afAl[0  , 0] := 1.00000E+01; afAl[0  , 1] := 2.70842E-02;
afAl[1  , 0] := 1.99800E+01; afAl[1  , 1] := 3.60106E-02;
afAl[2  , 0] := 2.99600E+01; afAl[2  , 1] := 1.04693E-01;
afAl[3  , 0] := 3.99400E+01; afAl[3  , 1] := 1.64797E-01;
afAl[4  , 0] := 4.99200E+01; afAl[4  , 1] := 1.89347E-01;
afAl[5  , 0] := 5.99000E+01; afAl[5  , 1] := 1.90141E-01;
afAl[6  , 0] := 6.98800E+01; afAl[6  , 1] := 1.82197E-01;
afAl[7  , 0] := 7.98600E+01; afAl[7  , 1] := 5.02769E+00;
afAl[8  , 0] := 8.98400E+01; afAl[8  , 1] := 6.70542E+00;
afAl[9  , 0] := 9.98200E+01; afAl[9  , 1] := 7.82345E+00;
afAl[10 , 0] := 1.09800E+02; afAl[10 , 1] := 8.42194E+00;
afAl[11 , 0] := 1.19780E+02; afAl[11 , 1] := 9.34640E+00;
afAl[12 , 0] := 1.29760E+02; afAl[12 , 1] := 9.38873E+00;
afAl[13 , 0] := 1.39740E+02; afAl[13 , 1] := 9.18537E+00;
afAl[14 , 0] := 1.49720E+02; afAl[14 , 1] := 8.86987E+00;
afAl[15 , 0] := 1.59700E+02; afAl[15 , 1] := 8.49608E+00;
afAl[16 , 0] := 1.69680E+02; afAl[16 , 1] := 8.09707E+00;
afAl[17 , 0] := 1.79660E+02; afAl[17 , 1] := 7.69477E+00;
afAl[18 , 0] := 1.89640E+02; afAl[18 , 1] := 7.30166E+00;
afAl[19 , 0] := 1.99620E+02; afAl[19 , 1] := 6.92482E+00;
afAl[20 , 0] := 2.09600E+02; afAl[20 , 1] := 6.56777E+00;
afAl[21 , 0] := 2.19580E+02; afAl[21 , 1] := 6.23207E+00;
afAl[22 , 0] := 2.29560E+02; afAl[22 , 1] := 5.91777E+00;
afAl[23 , 0] := 2.39540E+02; afAl[23 , 1] := 5.62454E+00;
afAl[24 , 0] := 2.49520E+02; afAl[24 , 1] := 5.35120E+00;
afAl[25 , 0] := 2.59500E+02; afAl[25 , 1] := 5.09661E+00;
afAl[26 , 0] := 2.69480E+02; afAl[26 , 1] := 4.85943E+00;
afAl[27 , 0] := 2.79460E+02; afAl[27 , 1] := 4.63835E+00;
afAl[28 , 0] := 2.89440E+02; afAl[28 , 1] := 4.43220E+00;
afAl[29 , 0] := 2.99420E+02; afAl[29 , 1] := 4.23955E+00;
afAl[30 , 0] := 3.09400E+02; afAl[30 , 1] := 4.05905E+00;
afAl[31 , 0] := 3.19380E+02; afAl[31 , 1] := 3.88982E+00;
afAl[32 , 0] := 3.29360E+02; afAl[32 , 1] := 3.73098E+00;
afAl[33 , 0] := 3.39340E+02; afAl[33 , 1] := 3.58176E+00;
afAl[34 , 0] := 3.49320E+02; afAl[34 , 1] := 3.44155E+00;
afAl[35 , 0] := 3.59300E+02; afAl[35 , 1] := 3.30950E+00;
afAl[36 , 0] := 3.69280E+02; afAl[36 , 1] := 3.18513E+00;
afAl[37 , 0] := 3.79260E+02; afAl[37 , 1] := 3.06777E+00;
afAl[38 , 0] := 3.89240E+02; afAl[38 , 1] := 2.95706E+00;
afAl[39 , 0] := 3.99220E+02; afAl[39 , 1] := 2.85236E+00;
afAl[40 , 0] := 4.09200E+02; afAl[40 , 1] := 2.75335E+00;
afAl[41 , 0] := 4.19180E+02; afAl[41 , 1] := 2.65961E+00;
afAl[42 , 0] := 4.29160E+02; afAl[42 , 1] := 2.57073E+00;
afAl[43 , 0] := 4.39140E+02; afAl[43 , 1] := 2.48642E+00;
afAl[44 , 0] := 4.49120E+02; afAl[44 , 1] := 2.40634E+00;
afAl[45 , 0] := 4.59100E+02; afAl[45 , 1] := 2.33034E+00;
afAl[46 , 0] := 4.69080E+02; afAl[46 , 1] := 2.25789E+00;
afAl[47 , 0] := 4.79060E+02; afAl[47 , 1] := 2.18898E+00;
afAl[48 , 0] := 4.89040E+02; afAl[48 , 1] := 2.12326E+00;
afAl[49 , 0] := 4.99020E+02; afAl[49 , 1] := 2.06057E+00;
afAl[50 , 0] := 5.09000E+02; afAl[50 , 1] := 2.00070E+00;
afAl[51 , 0] := 5.18980E+02; afAl[51 , 1] := 1.94346E+00;
afAl[52 , 0] := 5.28960E+02; afAl[52 , 1] := 1.88882E+00;
afAl[53 , 0] := 5.38940E+02; afAl[53 , 1] := 1.83643E+00;
afAl[54 , 0] := 5.48920E+02; afAl[54 , 1] := 1.78638E+00;
afAl[55 , 0] := 5.58900E+02; afAl[55 , 1] := 1.73837E+00;
afAl[56 , 0] := 5.68880E+02; afAl[56 , 1] := 1.69238E+00;
afAl[57 , 0] := 5.78860E+02; afAl[57 , 1] := 1.64824E+00;
afAl[58 , 0] := 5.88840E+02; afAl[58 , 1] := 1.60590E+00;
afAl[59 , 0] := 5.98820E+02; afAl[59 , 1] := 1.56527E+00;
afAl[60 , 0] := 6.08800E+02; afAl[60 , 1] := 1.52614E+00;
afAl[61 , 0] := 6.18780E+02; afAl[61 , 1] := 1.48866E+00;
afAl[62 , 0] := 6.28760E+02; afAl[62 , 1] := 1.45251E+00;
afAl[63 , 0] := 6.38740E+02; afAl[63 , 1] := 1.41780E+00;
afAl[64 , 0] := 6.48720E+02; afAl[64 , 1] := 1.38436E+00;
afAl[65 , 0] := 6.58700E+02; afAl[65 , 1] := 1.35214E+00;
afAl[66 , 0] := 6.68680E+02; afAl[66 , 1] := 1.32109E+00;
afAl[67 , 0] := 6.78660E+02; afAl[67 , 1] := 1.29118E+00;
afAl[68 , 0] := 6.88640E+02; afAl[68 , 1] := 1.26235E+00;
afAl[69 , 0] := 6.98620E+02; afAl[69 , 1] := 1.23455E+00;
afAl[70 , 0] := 7.08600E+02; afAl[70 , 1] := 1.20763E+00;
afAl[71 , 0] := 7.18580E+02; afAl[71 , 1] := 1.18169E+00;
afAl[72 , 0] := 7.28560E+02; afAl[72 , 1] := 1.15665E+00;
afAl[73 , 0] := 7.38540E+02; afAl[73 , 1] := 1.13241E+00;
afAl[74 , 0] := 7.48520E+02; afAl[74 , 1] := 1.10904E+00;
afAl[75 , 0] := 7.58500E+02; afAl[75 , 1] := 1.08635E+00;
afAl[76 , 0] := 7.68480E+02; afAl[76 , 1] := 1.06438E+00;
afAl[77 , 0] := 7.78460E+02; afAl[77 , 1] := 1.04320E+00;
afAl[78 , 0] := 7.88440E+02; afAl[78 , 1] := 1.02267E+00;
afAl[79 , 0] := 7.98420E+02; afAl[79 , 1] := 1.00279E+00;
afAl[80 , 0] := 8.08400E+02; afAl[80 , 1] := 9.83508E-01;
afAl[81 , 0] := 8.18380E+02; afAl[81 , 1] := 9.64827E-01;
afAl[82 , 0] := 8.28360E+02; afAl[82 , 1] := 9.46718E-01;
afAl[83 , 0] := 8.38340E+02; afAl[83 , 1] := 9.29156E-01;
afAl[84 , 0] := 8.48320E+02; afAl[84 , 1] := 9.12116E-01;
afAl[85 , 0] := 8.58300E+02; afAl[85 , 1] := 8.95580E-01;
afAl[86 , 0] := 8.68280E+02; afAl[86 , 1] := 8.79523E-01;
afAl[87 , 0] := 8.78260E+02; afAl[87 , 1] := 8.63940E-01;
afAl[88 , 0] := 8.88240E+02; afAl[88 , 1] := 8.48802E-01;
afAl[89 , 0] := 8.98220E+02; afAl[89 , 1] := 8.34091E-01;
afAl[90 , 0] := 9.08200E+02; afAl[90 , 1] := 8.19792E-01;
afAl[91 , 0] := 9.18180E+02; afAl[91 , 1] := 8.05893E-01;
afAl[92 , 0] := 9.28160E+02; afAl[92 , 1] := 7.92379E-01;
afAl[93 , 0] := 9.38140E+02; afAl[93 , 1] := 7.79238E-01;
afAl[94 , 0] := 9.48120E+02; afAl[94 , 1] := 7.66446E-01;
afAl[95 , 0] := 9.58100E+02; afAl[95 , 1] := 7.54006E-01;
afAl[96 , 0] := 9.68080E+02; afAl[96 , 1] := 7.41885E-01;
afAl[97 , 0] := 9.78060E+02; afAl[97 , 1] := 7.30099E-01;
afAl[98 , 0] := 9.88040E+02; afAl[98 , 1] := 7.18611E-01;
afAl[99 , 0] := 9.98020E+02; afAl[99 , 1] := 7.07387E-01;
afAl[100, 0] := 1.00800E+03; afAl[100, 1] := 6.95424E-01;
afAl[101, 0] := 1.01798E+03; afAl[101, 1] := 6.83488E-01;
afAl[102, 0] := 1.02796E+03; afAl[102, 1] := 6.71890E-01;
afAl[103, 0] := 1.03794E+03; afAl[103, 1] := 6.60613E-01;
afAl[104, 0] := 1.04792E+03; afAl[104, 1] := 6.49639E-01;
afAl[105, 0] := 1.05790E+03; afAl[105, 1] := 6.38961E-01;
afAl[106, 0] := 1.06788E+03; afAl[106, 1] := 6.28572E-01;
afAl[107, 0] := 1.07786E+03; afAl[107, 1] := 6.18448E-01;
afAl[108, 0] := 1.08784E+03; afAl[108, 1] := 6.08595E-01;
afAl[109, 0] := 1.09782E+03; afAl[109, 1] := 5.98997E-01;
afAl[110, 0] := 1.10780E+03; afAl[110, 1] := 5.89645E-01;
afAl[111, 0] := 1.11778E+03; afAl[111, 1] := 5.80527E-01;
afAl[112, 0] := 1.12776E+03; afAl[112, 1] := 5.71637E-01;
afAl[113, 0] := 1.13774E+03; afAl[113, 1] := 5.63091E-01;
afAl[114, 0] := 1.14772E+03; afAl[114, 1] := 5.55124E-01;
afAl[115, 0] := 1.15770E+03; afAl[115, 1] := 5.46894E-01;
afAl[116, 0] := 1.16768E+03; afAl[116, 1] := 5.38862E-01;
afAl[117, 0] := 1.17766E+03; afAl[117, 1] := 5.31030E-01;
afAl[118, 0] := 1.18764E+03; afAl[118, 1] := 5.23383E-01;
afAl[119, 0] := 1.19762E+03; afAl[119, 1] := 5.15914E-01;
afAl[120, 0] := 1.20760E+03; afAl[120, 1] := 5.08620E-01;
afAl[121, 0] := 1.21758E+03; afAl[121, 1] := 5.01502E-01;
afAl[122, 0] := 1.22756E+03; afAl[122, 1] := 4.94552E-01;
afAl[123, 0] := 1.23754E+03; afAl[123, 1] := 4.87758E-01;
afAl[124, 0] := 1.24752E+03; afAl[124, 1] := 4.81121E-01;
afAl[125, 0] := 1.25750E+03; afAl[125, 1] := 4.74634E-01;
afAl[126, 0] := 1.26748E+03; afAl[126, 1] := 4.68288E-01;
afAl[127, 0] := 1.27746E+03; afAl[127, 1] := 4.62094E-01;
afAl[128, 0] := 1.28744E+03; afAl[128, 1] := 4.56035E-01;
afAl[129, 0] := 1.29742E+03; afAl[129, 1] := 4.50111E-01;
afAl[130, 0] := 1.30740E+03; afAl[130, 1] := 4.44316E-01;
afAl[131, 0] := 1.31738E+03; afAl[131, 1] := 4.38642E-01;
afAl[132, 0] := 1.32736E+03; afAl[132, 1] := 4.33101E-01;
afAl[133, 0] := 1.33734E+03; afAl[133, 1] := 4.27680E-01;
afAl[134, 0] := 1.34732E+03; afAl[134, 1] := 4.22377E-01;
afAl[135, 0] := 1.35730E+03; afAl[135, 1] := 4.17190E-01;
afAl[136, 0] := 1.36728E+03; afAl[136, 1] := 4.12113E-01;
afAl[137, 0] := 1.37726E+03; afAl[137, 1] := 4.07019E-01;
afAl[138, 0] := 1.38724E+03; afAl[138, 1] := 4.01929E-01;
afAl[139, 0] := 1.39722E+03; afAl[139, 1] := 3.96949E-01;
afAl[140, 0] := 1.40720E+03; afAl[140, 1] := 3.92089E-01;
afAl[141, 0] := 1.41718E+03; afAl[141, 1] := 3.87341E-01;
afAl[142, 0] := 1.42716E+03; afAl[142, 1] := 3.82702E-01;
afAl[143, 0] := 1.43714E+03; afAl[143, 1] := 3.78198E-01;
afAl[144, 0] := 1.44712E+03; afAl[144, 1] := 3.73809E-01;
afAl[145, 0] := 1.45710E+03; afAl[145, 1] := 3.69535E-01;
afAl[146, 0] := 1.46708E+03; afAl[146, 1] := 3.65412E-01;
afAl[147, 0] := 1.47706E+03; afAl[147, 1] := 3.61445E-01;
afAl[148, 0] := 1.48704E+03; afAl[148, 1] := 3.57628E-01;
afAl[149, 0] := 1.49702E+03; afAl[149, 1] := 3.54048E-01;
afAl[150, 0] := 1.50700E+03; afAl[150, 1] := 3.50804E-01;
afAl[151, 0] := 1.51698E+03; afAl[151, 1] := 3.47914E-01;
afAl[152, 0] := 1.52696E+03; afAl[152, 1] := 3.45929E-01;
afAl[153, 0] := 1.53694E+03; afAl[153, 1] := 3.46742E-01;
afAl[154, 0] := 1.54692E+03; afAl[154, 1] := 3.50697E-01;
afAl[155, 0] := 1.55690E+03; afAl[155, 1] := 4.26944E-01;
afAl[156, 0] := 1.56688E+03; afAl[156, 1] := 4.02112E+00;
afAl[157, 0] := 1.57686E+03; afAl[157, 1] := 4.03269E+00;
afAl[158, 0] := 1.58684E+03; afAl[158, 1] := 4.02760E+00;
afAl[159, 0] := 1.59682E+03; afAl[159, 1] := 4.02146E+00;
afAl[160, 0] := 1.60680E+03; afAl[160, 1] := 4.01388E+00;
afAl[161, 0] := 1.61678E+03; afAl[161, 1] := 4.00574E+00;
afAl[162, 0] := 1.62676E+03; afAl[162, 1] := 3.99650E+00;
afAl[163, 0] := 1.63674E+03; afAl[163, 1] := 3.98341E+00;
afAl[164, 0] := 1.64672E+03; afAl[164, 1] := 3.96271E+00;
afAl[165, 0] := 1.65670E+03; afAl[165, 1] := 3.93665E+00;
afAl[166, 0] := 1.66668E+03; afAl[166, 1] := 3.90900E+00;
afAl[167, 0] := 1.67666E+03; afAl[167, 1] := 3.88107E+00;
afAl[168, 0] := 1.68664E+03; afAl[168, 1] := 3.85213E+00;
afAl[169, 0] := 1.69662E+03; afAl[169, 1] := 3.82264E+00;
afAl[170, 0] := 1.70660E+03; afAl[170, 1] := 3.79294E+00;
afAl[171, 0] := 1.71658E+03; afAl[171, 1] := 3.76227E+00;
afAl[172, 0] := 1.72656E+03; afAl[172, 1] := 3.73163E+00;
afAl[173, 0] := 1.73654E+03; afAl[173, 1] := 3.70036E+00;
afAl[174, 0] := 1.74652E+03; afAl[174, 1] := 3.66898E+00;
afAl[175, 0] := 1.75650E+03; afAl[175, 1] := 3.63739E+00;
afAl[176, 0] := 1.76648E+03; afAl[176, 1] := 3.60559E+00;
afAl[177, 0] := 1.77646E+03; afAl[177, 1] := 3.57397E+00;
afAl[178, 0] := 1.78644E+03; afAl[178, 1] := 3.54191E+00;
afAl[179, 0] := 1.79642E+03; afAl[179, 1] := 3.51015E+00;
afAl[180, 0] := 1.80640E+03; afAl[180, 1] := 3.47823E+00;
afAl[181, 0] := 1.81638E+03; afAl[181, 1] := 3.44653E+00;
afAl[182, 0] := 1.82636E+03; afAl[182, 1] := 3.41485E+00;
afAl[183, 0] := 1.83634E+03; afAl[183, 1] := 3.38331E+00;
afAl[184, 0] := 1.84632E+03; afAl[184, 1] := 3.35198E+00;
afAl[185, 0] := 1.85630E+03; afAl[185, 1] := 3.32076E+00;
afAl[186, 0] := 1.86628E+03; afAl[186, 1] := 3.28986E+00;
afAl[187, 0] := 1.87626E+03; afAl[187, 1] := 3.25914E+00;
afAl[188, 0] := 1.88624E+03; afAl[188, 1] := 3.22882E+00;
afAl[189, 0] := 1.89622E+03; afAl[189, 1] := 3.19857E+00;
afAl[190, 0] := 1.90620E+03; afAl[190, 1] := 3.16874E+00;
afAl[191, 0] := 1.91618E+03; afAl[191, 1] := 3.13915E+00;
afAl[192, 0] := 1.92616E+03; afAl[192, 1] := 3.10995E+00;
afAl[193, 0] := 1.93614E+03; afAl[193, 1] := 3.08100E+00;
afAl[194, 0] := 1.94612E+03; afAl[194, 1] := 3.05244E+00;
afAl[195, 0] := 1.95610E+03; afAl[195, 1] := 3.02422E+00;
afAl[196, 0] := 1.96608E+03; afAl[196, 1] := 2.99638E+00;
afAl[197, 0] := 1.97606E+03; afAl[197, 1] := 2.96892E+00;
afAl[198, 0] := 1.98604E+03; afAl[198, 1] := 2.94192E+00;
afAl[199, 0] := 1.99602E+03; afAl[199, 1] := 2.91544E+00;
afAl[200, 0] := 2.00600E+03; afAl[200, 1] := 2.88923E+00;
afAl[201, 0] := 2.01598E+03; afAl[201, 1] := 2.86321E+00;
afAl[202, 0] := 2.02596E+03; afAl[202, 1] := 2.83810E+00;
afAl[203, 0] := 2.03594E+03; afAl[203, 1] := 2.81427E+00;
afAl[204, 0] := 2.04592E+03; afAl[204, 1] := 2.79094E+00;
afAl[205, 0] := 2.05590E+03; afAl[205, 1] := 2.76826E+00;
afAl[206, 0] := 2.06588E+03; afAl[206, 1] := 2.74590E+00;
afAl[207, 0] := 2.07586E+03; afAl[207, 1] := 2.72387E+00;
afAl[208, 0] := 2.08584E+03; afAl[208, 1] := 2.70213E+00;
afAl[209, 0] := 2.09582E+03; afAl[209, 1] := 2.68073E+00;
afAl[210, 0] := 2.10580E+03; afAl[210, 1] := 2.65961E+00;
afAl[211, 0] := 2.11578E+03; afAl[211, 1] := 2.63883E+00;
afAl[212, 0] := 2.12576E+03; afAl[212, 1] := 2.61831E+00;
afAl[213, 0] := 2.13574E+03; afAl[213, 1] := 2.59812E+00;
afAl[214, 0] := 2.14572E+03; afAl[214, 1] := 2.57819E+00;
afAl[215, 0] := 2.15570E+03; afAl[215, 1] := 2.55859E+00;
afAl[216, 0] := 2.16568E+03; afAl[216, 1] := 2.53923E+00;
afAl[217, 0] := 2.17566E+03; afAl[217, 1] := 2.52012E+00;
afAl[218, 0] := 2.18564E+03; afAl[218, 1] := 2.50124E+00;
afAl[219, 0] := 2.19562E+03; afAl[219, 1] := 2.48265E+00;
afAl[220, 0] := 2.20560E+03; afAl[220, 1] := 2.46432E+00;
afAl[221, 0] := 2.21558E+03; afAl[221, 1] := 2.44619E+00;
afAl[222, 0] := 2.22556E+03; afAl[222, 1] := 2.42823E+00;
afAl[223, 0] := 2.23554E+03; afAl[223, 1] := 2.41049E+00;
afAl[224, 0] := 2.24552E+03; afAl[224, 1] := 2.39302E+00;
afAl[225, 0] := 2.25550E+03; afAl[225, 1] := 2.37575E+00;
afAl[226, 0] := 2.26548E+03; afAl[226, 1] := 2.35871E+00;
afAl[227, 0] := 2.27546E+03; afAl[227, 1] := 2.34188E+00;
afAl[228, 0] := 2.28544E+03; afAl[228, 1] := 2.32525E+00;
afAl[229, 0] := 2.29542E+03; afAl[229, 1] := 2.30884E+00;
afAl[230, 0] := 2.30540E+03; afAl[230, 1] := 2.29262E+00;
afAl[231, 0] := 2.31538E+03; afAl[231, 1] := 2.27662E+00;
afAl[232, 0] := 2.32536E+03; afAl[232, 1] := 2.26079E+00;
afAl[233, 0] := 2.33534E+03; afAl[233, 1] := 2.24515E+00;
afAl[234, 0] := 2.34532E+03; afAl[234, 1] := 2.22968E+00;
afAl[235, 0] := 2.35530E+03; afAl[235, 1] := 2.21442E+00;
afAl[236, 0] := 2.36528E+03; afAl[236, 1] := 2.19934E+00;
afAl[237, 0] := 2.37526E+03; afAl[237, 1] := 2.18443E+00;
afAl[238, 0] := 2.38524E+03; afAl[238, 1] := 2.16970E+00;
afAl[239, 0] := 2.39522E+03; afAl[239, 1] := 2.15513E+00;
afAl[240, 0] := 2.40520E+03; afAl[240, 1] := 2.14077E+00;
afAl[241, 0] := 2.41518E+03; afAl[241, 1] := 2.12657E+00;
afAl[242, 0] := 2.42516E+03; afAl[242, 1] := 2.11251E+00;
afAl[243, 0] := 2.43514E+03; afAl[243, 1] := 2.09859E+00;
afAl[244, 0] := 2.44512E+03; afAl[244, 1] := 2.08482E+00;
afAl[245, 0] := 2.45510E+03; afAl[245, 1] := 2.07118E+00;
afAl[246, 0] := 2.46508E+03; afAl[246, 1] := 2.05769E+00;
afAl[247, 0] := 2.47506E+03; afAl[247, 1] := 2.04436E+00;
afAl[248, 0] := 2.48504E+03; afAl[248, 1] := 2.03118E+00;
afAl[249, 0] := 2.49502E+03; afAl[249, 1] := 2.01813E+00;
afAl[250, 0] := 2.50500E+03; afAl[250, 1] := 2.00521E+00;
afAl[251, 0] := 2.51498E+03; afAl[251, 1] := 1.99243E+00;
afAl[252, 0] := 2.52496E+03; afAl[252, 1] := 1.97980E+00;
afAl[253, 0] := 2.53494E+03; afAl[253, 1] := 1.96732E+00;
afAl[254, 0] := 2.54492E+03; afAl[254, 1] := 1.95495E+00;
afAl[255, 0] := 2.55490E+03; afAl[255, 1] := 1.94268E+00;
afAl[256, 0] := 2.56488E+03; afAl[256, 1] := 1.93053E+00;
afAl[257, 0] := 2.57486E+03; afAl[257, 1] := 1.91850E+00;
afAl[258, 0] := 2.58484E+03; afAl[258, 1] := 1.90660E+00;
afAl[259, 0] := 2.59482E+03; afAl[259, 1] := 1.89482E+00;
afAl[260, 0] := 2.60480E+03; afAl[260, 1] := 1.88316E+00;
afAl[261, 0] := 2.61478E+03; afAl[261, 1] := 1.87162E+00;
afAl[262, 0] := 2.62476E+03; afAl[262, 1] := 1.86019E+00;
afAl[263, 0] := 2.63474E+03; afAl[263, 1] := 1.84888E+00;
afAl[264, 0] := 2.64472E+03; afAl[264, 1] := 1.83769E+00;
afAl[265, 0] := 2.65470E+03; afAl[265, 1] := 1.82654E+00;
afAl[266, 0] := 2.66468E+03; afAl[266, 1] := 1.81550E+00;
afAl[267, 0] := 2.67466E+03; afAl[267, 1] := 1.80457E+00;
afAl[268, 0] := 2.68464E+03; afAl[268, 1] := 1.79380E+00;
afAl[269, 0] := 2.69462E+03; afAl[269, 1] := 1.78312E+00;
afAl[270, 0] := 2.70460E+03; afAl[270, 1] := 1.77251E+00;
afAl[271, 0] := 2.71458E+03; afAl[271, 1] := 1.76198E+00;
afAl[272, 0] := 2.72456E+03; afAl[272, 1] := 1.75156E+00;
afAl[273, 0] := 2.73454E+03; afAl[273, 1] := 1.74124E+00;
afAl[274, 0] := 2.74452E+03; afAl[274, 1] := 1.73103E+00;
afAl[275, 0] := 2.75450E+03; afAl[275, 1] := 1.72091E+00;
afAl[276, 0] := 2.76448E+03; afAl[276, 1] := 1.71087E+00;
afAl[277, 0] := 2.77446E+03; afAl[277, 1] := 1.70093E+00;
afAl[278, 0] := 2.78444E+03; afAl[278, 1] := 1.69107E+00;
afAl[279, 0] := 2.79442E+03; afAl[279, 1] := 1.68130E+00;
afAl[280, 0] := 2.80440E+03; afAl[280, 1] := 1.67162E+00;
afAl[281, 0] := 2.81438E+03; afAl[281, 1] := 1.66200E+00;
afAl[282, 0] := 2.82436E+03; afAl[282, 1] := 1.65245E+00;
afAl[283, 0] := 2.83434E+03; afAl[283, 1] := 1.64298E+00;
afAl[284, 0] := 2.84432E+03; afAl[284, 1] := 1.63363E+00;
afAl[285, 0] := 2.85430E+03; afAl[285, 1] := 1.62436E+00;
afAl[286, 0] := 2.86428E+03; afAl[286, 1] := 1.61518E+00;
afAl[287, 0] := 2.87426E+03; afAl[287, 1] := 1.60608E+00;
afAl[288, 0] := 2.88424E+03; afAl[288, 1] := 1.59706E+00;
afAl[289, 0] := 2.89422E+03; afAl[289, 1] := 1.58812E+00;
afAl[290, 0] := 2.90420E+03; afAl[290, 1] := 1.57922E+00;
afAl[291, 0] := 2.91418E+03; afAl[291, 1] := 1.57040E+00;
afAl[292, 0] := 2.92416E+03; afAl[292, 1] := 1.56166E+00;
afAl[293, 0] := 2.93414E+03; afAl[293, 1] := 1.55299E+00;
afAl[294, 0] := 2.94412E+03; afAl[294, 1] := 1.54440E+00;
afAl[295, 0] := 2.95410E+03; afAl[295, 1] := 1.53589E+00;
afAl[296, 0] := 2.96408E+03; afAl[296, 1] := 1.52745E+00;
afAl[297, 0] := 2.97406E+03; afAl[297, 1] := 1.51908E+00;
afAl[298, 0] := 2.98404E+03; afAl[298, 1] := 1.51074E+00;
afAl[299, 0] := 2.99402E+03; afAl[299, 1] := 1.50235E+00;
afAl[300, 0] := 3.00400E+03; afAl[300, 1] := 1.49404E+00;
afAl[301, 0] := 3.01398E+03; afAl[301, 1] := 1.48573E+00;
afAl[302, 0] := 3.02396E+03; afAl[302, 1] := 1.47732E+00;
afAl[303, 0] := 3.03394E+03; afAl[303, 1] := 1.46899E+00;
afAl[304, 0] := 3.04392E+03; afAl[304, 1] := 1.46074E+00;
afAl[305, 0] := 3.05390E+03; afAl[305, 1] := 1.45258E+00;
afAl[306, 0] := 3.06388E+03; afAl[306, 1] := 1.44450E+00;
afAl[307, 0] := 3.07386E+03; afAl[307, 1] := 1.43647E+00;
afAl[308, 0] := 3.08384E+03; afAl[308, 1] := 1.42849E+00;
afAl[309, 0] := 3.09382E+03; afAl[309, 1] := 1.42057E+00;
afAl[310, 0] := 3.10380E+03; afAl[310, 1] := 1.41270E+00;
afAl[311, 0] := 3.11378E+03; afAl[311, 1] := 1.40476E+00;
afAl[312, 0] := 3.12376E+03; afAl[312, 1] := 1.39688E+00;
afAl[313, 0] := 3.13374E+03; afAl[313, 1] := 1.38906E+00;
afAl[314, 0] := 3.14372E+03; afAl[314, 1] := 1.38103E+00;
afAl[315, 0] := 3.15370E+03; afAl[315, 1] := 1.37306E+00;
afAl[316, 0] := 3.16368E+03; afAl[316, 1] := 1.36517E+00;
afAl[317, 0] := 3.17366E+03; afAl[317, 1] := 1.35733E+00;
afAl[318, 0] := 3.18364E+03; afAl[318, 1] := 1.34956E+00;
afAl[319, 0] := 3.19362E+03; afAl[319, 1] := 1.34186E+00;
afAl[320, 0] := 3.20360E+03; afAl[320, 1] := 1.33427E+00;
afAl[321, 0] := 3.21358E+03; afAl[321, 1] := 1.32675E+00;
afAl[322, 0] := 3.22356E+03; afAl[322, 1] := 1.31930E+00;
afAl[323, 0] := 3.23354E+03; afAl[323, 1] := 1.31189E+00;
afAl[324, 0] := 3.24352E+03; afAl[324, 1] := 1.30452E+00;
afAl[325, 0] := 3.25350E+03; afAl[325, 1] := 1.29722E+00;
afAl[326, 0] := 3.26348E+03; afAl[326, 1] := 1.28999E+00;
afAl[327, 0] := 3.27346E+03; afAl[327, 1] := 1.28284E+00;
afAl[328, 0] := 3.28344E+03; afAl[328, 1] := 1.27575E+00;
afAl[329, 0] := 3.29342E+03; afAl[329, 1] := 1.26872E+00;
afAl[330, 0] := 3.30340E+03; afAl[330, 1] := 1.26175E+00;
afAl[331, 0] := 3.31338E+03; afAl[331, 1] := 1.25483E+00;
afAl[332, 0] := 3.32336E+03; afAl[332, 1] := 1.24797E+00;
afAl[333, 0] := 3.33334E+03; afAl[333, 1] := 1.24117E+00;
afAl[334, 0] := 3.34332E+03; afAl[334, 1] := 1.23443E+00;
afAl[335, 0] := 3.35330E+03; afAl[335, 1] := 1.22774E+00;
afAl[336, 0] := 3.36328E+03; afAl[336, 1] := 1.22110E+00;
afAl[337, 0] := 3.37326E+03; afAl[337, 1] := 1.21453E+00;
afAl[338, 0] := 3.38324E+03; afAl[338, 1] := 1.20800E+00;
afAl[339, 0] := 3.39322E+03; afAl[339, 1] := 1.20153E+00;
afAl[340, 0] := 3.40320E+03; afAl[340, 1] := 1.19512E+00;
afAl[341, 0] := 3.41318E+03; afAl[341, 1] := 1.18876E+00;
afAl[342, 0] := 3.42316E+03; afAl[342, 1] := 1.18245E+00;
afAl[343, 0] := 3.43314E+03; afAl[343, 1] := 1.17619E+00;
afAl[344, 0] := 3.44312E+03; afAl[344, 1] := 1.16999E+00;
afAl[345, 0] := 3.45310E+03; afAl[345, 1] := 1.16384E+00;
afAl[346, 0] := 3.46308E+03; afAl[346, 1] := 1.15773E+00;
afAl[347, 0] := 3.47306E+03; afAl[347, 1] := 1.15169E+00;
afAl[348, 0] := 3.48304E+03; afAl[348, 1] := 1.14569E+00;
afAl[349, 0] := 3.49302E+03; afAl[349, 1] := 1.13974E+00;
afAl[350, 0] := 3.50300E+03; afAl[350, 1] := 1.13382E+00;
afAl[351, 0] := 3.51298E+03; afAl[351, 1] := 1.12794E+00;
afAl[352, 0] := 3.52296E+03; afAl[352, 1] := 1.12211E+00;
afAl[353, 0] := 3.53294E+03; afAl[353, 1] := 1.11634E+00;
afAl[354, 0] := 3.54292E+03; afAl[354, 1] := 1.11064E+00;
afAl[355, 0] := 3.55290E+03; afAl[355, 1] := 1.10498E+00;
afAl[356, 0] := 3.56288E+03; afAl[356, 1] := 1.09937E+00;
afAl[357, 0] := 3.57286E+03; afAl[357, 1] := 1.09378E+00;
afAl[358, 0] := 3.58284E+03; afAl[358, 1] := 1.08821E+00;
afAl[359, 0] := 3.59282E+03; afAl[359, 1] := 1.08269E+00;
afAl[360, 0] := 3.60280E+03; afAl[360, 1] := 1.07721E+00;
afAl[361, 0] := 3.61278E+03; afAl[361, 1] := 1.07181E+00;
afAl[362, 0] := 3.62276E+03; afAl[362, 1] := 1.06646E+00;
afAl[363, 0] := 3.63274E+03; afAl[363, 1] := 1.06114E+00;
afAl[364, 0] := 3.64272E+03; afAl[364, 1] := 1.05587E+00;
afAl[365, 0] := 3.65270E+03; afAl[365, 1] := 1.05062E+00;
afAl[366, 0] := 3.66268E+03; afAl[366, 1] := 1.04542E+00;
afAl[367, 0] := 3.67266E+03; afAl[367, 1] := 1.04025E+00;
afAl[368, 0] := 3.68264E+03; afAl[368, 1] := 1.03512E+00;
afAl[369, 0] := 3.69262E+03; afAl[369, 1] := 1.03002E+00;
afAl[370, 0] := 3.70260E+03; afAl[370, 1] := 1.02496E+00;
afAl[371, 0] := 3.71258E+03; afAl[371, 1] := 1.01994E+00;
afAl[372, 0] := 3.72256E+03; afAl[372, 1] := 1.01498E+00;
afAl[373, 0] := 3.73254E+03; afAl[373, 1] := 1.01005E+00;
afAl[374, 0] := 3.74252E+03; afAl[374, 1] := 1.00516E+00;
afAl[375, 0] := 3.75250E+03; afAl[375, 1] := 1.00029E+00;
afAl[376, 0] := 3.76248E+03; afAl[376, 1] := 9.95458E-01;
afAl[377, 0] := 3.77246E+03; afAl[377, 1] := 9.90658E-01;
afAl[378, 0] := 3.78244E+03; afAl[378, 1] := 9.85893E-01;
afAl[379, 0] := 3.79242E+03; afAl[379, 1] := 9.81173E-01;
afAl[380, 0] := 3.80240E+03; afAl[380, 1] := 9.76491E-01;
afAl[381, 0] := 3.81238E+03; afAl[381, 1] := 9.71843E-01;
afAl[382, 0] := 3.82236E+03; afAl[382, 1] := 9.67230E-01;
afAl[383, 0] := 3.83234E+03; afAl[383, 1] := 9.62646E-01;
afAl[384, 0] := 3.84232E+03; afAl[384, 1] := 9.58096E-01;
afAl[385, 0] := 3.85230E+03; afAl[385, 1] := 9.53579E-01;
afAl[386, 0] := 3.86228E+03; afAl[386, 1] := 9.49094E-01;
afAl[387, 0] := 3.87226E+03; afAl[387, 1] := 9.44645E-01;
afAl[388, 0] := 3.88224E+03; afAl[388, 1] := 9.40227E-01;
afAl[389, 0] := 3.89222E+03; afAl[389, 1] := 9.35842E-01;
afAl[390, 0] := 3.90220E+03; afAl[390, 1] := 9.31488E-01;
afAl[391, 0] := 3.91218E+03; afAl[391, 1] := 9.27167E-01;
afAl[392, 0] := 3.92216E+03; afAl[392, 1] := 9.22876E-01;
afAl[393, 0] := 3.93214E+03; afAl[393, 1] := 9.18616E-01;
afAl[394, 0] := 3.94212E+03; afAl[394, 1] := 9.14386E-01;
afAl[395, 0] := 3.95210E+03; afAl[395, 1] := 9.10183E-01;
afAl[396, 0] := 3.96208E+03; afAl[396, 1] := 9.06011E-01;
afAl[397, 0] := 3.97206E+03; afAl[397, 1] := 9.01868E-01;
afAl[398, 0] := 3.98204E+03; afAl[398, 1] := 8.97756E-01;
afAl[399, 0] := 3.99202E+03; afAl[399, 1] := 8.93675E-01;
afAl[400, 0] := 4.00200E+03; afAl[400, 1] := 8.89623E-01;
afAl[401, 0] := 4.01198E+03; afAl[401, 1] := 8.85599E-01;
afAl[402, 0] := 4.02196E+03; afAl[402, 1] := 8.81603E-01;
afAl[403, 0] := 4.03194E+03; afAl[403, 1] := 8.77633E-01;
afAl[404, 0] := 4.04192E+03; afAl[404, 1] := 8.73690E-01;
afAl[405, 0] := 4.05190E+03; afAl[405, 1] := 8.69775E-01;
afAl[406, 0] := 4.06188E+03; afAl[406, 1] := 8.65887E-01;
afAl[407, 0] := 4.07186E+03; afAl[407, 1] := 8.62027E-01;
afAl[408, 0] := 4.08184E+03; afAl[408, 1] := 8.58194E-01;
afAl[409, 0] := 4.09182E+03; afAl[409, 1] := 8.54387E-01;
afAl[410, 0] := 4.10180E+03; afAl[410, 1] := 8.50606E-01;
afAl[411, 0] := 4.11178E+03; afAl[411, 1] := 8.46851E-01;
afAl[412, 0] := 4.12176E+03; afAl[412, 1] := 8.43122E-01;
afAl[413, 0] := 4.13174E+03; afAl[413, 1] := 8.39418E-01;
afAl[414, 0] := 4.14172E+03; afAl[414, 1] := 8.35739E-01;
afAl[415, 0] := 4.15170E+03; afAl[415, 1] := 8.32087E-01;
afAl[416, 0] := 4.16168E+03; afAl[416, 1] := 8.28459E-01;
afAl[417, 0] := 4.17166E+03; afAl[417, 1] := 8.24856E-01;
afAl[418, 0] := 4.18164E+03; afAl[418, 1] := 8.21276E-01;
afAl[419, 0] := 4.19162E+03; afAl[419, 1] := 8.17721E-01;
afAl[420, 0] := 4.20160E+03; afAl[420, 1] := 8.14190E-01;
afAl[421, 0] := 4.21158E+03; afAl[421, 1] := 8.10683E-01;
afAl[422, 0] := 4.22156E+03; afAl[422, 1] := 8.07198E-01;
afAl[423, 0] := 4.23154E+03; afAl[423, 1] := 8.03736E-01;
afAl[424, 0] := 4.24152E+03; afAl[424, 1] := 8.00297E-01;
afAl[425, 0] := 4.25150E+03; afAl[425, 1] := 7.96880E-01;
afAl[426, 0] := 4.26148E+03; afAl[426, 1] := 7.93486E-01;
afAl[427, 0] := 4.27146E+03; afAl[427, 1] := 7.90115E-01;
afAl[428, 0] := 4.28144E+03; afAl[428, 1] := 7.86765E-01;
afAl[429, 0] := 4.29142E+03; afAl[429, 1] := 7.83438E-01;
afAl[430, 0] := 4.30140E+03; afAl[430, 1] := 7.80132E-01;
afAl[431, 0] := 4.31138E+03; afAl[431, 1] := 7.76848E-01;
afAl[432, 0] := 4.32136E+03; afAl[432, 1] := 7.73586E-01;
afAl[433, 0] := 4.33134E+03; afAl[433, 1] := 7.70346E-01;
afAl[434, 0] := 4.34132E+03; afAl[434, 1] := 7.67126E-01;
afAl[435, 0] := 4.35130E+03; afAl[435, 1] := 7.63928E-01;
afAl[436, 0] := 4.36128E+03; afAl[436, 1] := 7.60749E-01;
afAl[437, 0] := 4.37126E+03; afAl[437, 1] := 7.57592E-01;
afAl[438, 0] := 4.38124E+03; afAl[438, 1] := 7.54454E-01;
afAl[439, 0] := 4.39122E+03; afAl[439, 1] := 7.51337E-01;
afAl[440, 0] := 4.40120E+03; afAl[440, 1] := 7.48238E-01;
afAl[441, 0] := 4.41118E+03; afAl[441, 1] := 7.45159E-01;
afAl[442, 0] := 4.42116E+03; afAl[442, 1] := 7.42099E-01;
afAl[443, 0] := 4.43114E+03; afAl[443, 1] := 7.39059E-01;
afAl[444, 0] := 4.44112E+03; afAl[444, 1] := 7.36039E-01;
afAl[445, 0] := 4.45110E+03; afAl[445, 1] := 7.33039E-01;
afAl[446, 0] := 4.46108E+03; afAl[446, 1] := 7.30058E-01;
afAl[447, 0] := 4.47106E+03; afAl[447, 1] := 7.27095E-01;
afAl[448, 0] := 4.48104E+03; afAl[448, 1] := 7.24152E-01;
afAl[449, 0] := 4.49102E+03; afAl[449, 1] := 7.21227E-01;
afAl[450, 0] := 4.50100E+03; afAl[450, 1] := 7.18320E-01;
afAl[451, 0] := 4.51098E+03; afAl[451, 1] := 7.15432E-01;
afAl[452, 0] := 4.52096E+03; afAl[452, 1] := 7.12562E-01;
afAl[453, 0] := 4.53094E+03; afAl[453, 1] := 7.09709E-01;
afAl[454, 0] := 4.54092E+03; afAl[454, 1] := 7.06874E-01;
afAl[455, 0] := 4.55090E+03; afAl[455, 1] := 7.04056E-01;
afAl[456, 0] := 4.56088E+03; afAl[456, 1] := 7.01255E-01;
afAl[457, 0] := 4.57086E+03; afAl[457, 1] := 6.98472E-01;
afAl[458, 0] := 4.58084E+03; afAl[458, 1] := 6.95705E-01;
afAl[459, 0] := 4.59082E+03; afAl[459, 1] := 6.92956E-01;
afAl[460, 0] := 4.60080E+03; afAl[460, 1] := 6.90224E-01;
afAl[461, 0] := 4.61078E+03; afAl[461, 1] := 6.87508E-01;
afAl[462, 0] := 4.62076E+03; afAl[462, 1] := 6.84809E-01;
afAl[463, 0] := 4.63074E+03; afAl[463, 1] := 6.82125E-01;
afAl[464, 0] := 4.64072E+03; afAl[464, 1] := 6.79458E-01;
afAl[465, 0] := 4.65070E+03; afAl[465, 1] := 6.76806E-01;
afAl[466, 0] := 4.66068E+03; afAl[466, 1] := 6.74171E-01;
afAl[467, 0] := 4.67066E+03; afAl[467, 1] := 6.71553E-01;
afAl[468, 0] := 4.68064E+03; afAl[468, 1] := 6.68951E-01;
afAl[469, 0] := 4.69062E+03; afAl[469, 1] := 6.66365E-01;
afAl[470, 0] := 4.70060E+03; afAl[470, 1] := 6.63794E-01;
afAl[471, 0] := 4.71058E+03; afAl[471, 1] := 6.61239E-01;
afAl[472, 0] := 4.72056E+03; afAl[472, 1] := 6.58697E-01;
afAl[473, 0] := 4.73054E+03; afAl[473, 1] := 6.56171E-01;
afAl[474, 0] := 4.74052E+03; afAl[474, 1] := 6.53659E-01;
afAl[475, 0] := 4.75050E+03; afAl[475, 1] := 6.51163E-01;
afAl[476, 0] := 4.76048E+03; afAl[476, 1] := 6.48681E-01;
afAl[477, 0] := 4.77046E+03; afAl[477, 1] := 6.46216E-01;
afAl[478, 0] := 4.78044E+03; afAl[478, 1] := 6.43764E-01;
afAl[479, 0] := 4.79042E+03; afAl[479, 1] := 6.41328E-01;
afAl[480, 0] := 4.80040E+03; afAl[480, 1] := 6.38905E-01;
afAl[481, 0] := 4.81038E+03; afAl[481, 1] := 6.36497E-01;
afAl[482, 0] := 4.82036E+03; afAl[482, 1] := 6.34103E-01;
afAl[483, 0] := 4.83034E+03; afAl[483, 1] := 6.31723E-01;
afAl[484, 0] := 4.84032E+03; afAl[484, 1] := 6.29356E-01;
afAl[485, 0] := 4.85030E+03; afAl[485, 1] := 6.27004E-01;
afAl[486, 0] := 4.86028E+03; afAl[486, 1] := 6.24664E-01;
afAl[487, 0] := 4.87026E+03; afAl[487, 1] := 6.22338E-01;
afAl[488, 0] := 4.88024E+03; afAl[488, 1] := 6.20024E-01;
afAl[489, 0] := 4.89022E+03; afAl[489, 1] := 6.17725E-01;
afAl[490, 0] := 4.90020E+03; afAl[490, 1] := 6.15438E-01;
afAl[491, 0] := 4.91018E+03; afAl[491, 1] := 6.13164E-01;
afAl[492, 0] := 4.92016E+03; afAl[492, 1] := 6.10903E-01;
afAl[493, 0] := 4.93014E+03; afAl[493, 1] := 6.08655E-01;
afAl[494, 0] := 4.94012E+03; afAl[494, 1] := 6.06420E-01;
afAl[495, 0] := 4.95010E+03; afAl[495, 1] := 6.04198E-01;
afAl[496, 0] := 4.96008E+03; afAl[496, 1] := 6.01988E-01;
afAl[497, 0] := 4.97006E+03; afAl[497, 1] := 5.99791E-01;
afAl[498, 0] := 4.98004E+03; afAl[498, 1] := 5.97607E-01;
afAl[499, 0] := 4.99002E+03; afAl[499, 1] := 5.95434E-01;
afAl[500, 0] := 5.00000E+03; afAl[500, 1] := 5.93274E-01;
afAl[501, 0] := 5.05000E+03; afAl[501, 1] := 5.82639E-01;
afAl[502, 0] := 5.10000E+03; afAl[502, 1] := 5.72295E-01;
afAl[503, 0] := 5.15000E+03; afAl[503, 1] := 5.62227E-01;
afAl[504, 0] := 5.20000E+03; afAl[504, 1] := 5.52436E-01;
afAl[505, 0] := 5.25000E+03; afAl[505, 1] := 5.42906E-01;
afAl[506, 0] := 5.30000E+03; afAl[506, 1] := 5.33631E-01;
afAl[507, 0] := 5.35000E+03; afAl[507, 1] := 5.24597E-01;
afAl[508, 0] := 5.40000E+03; afAl[508, 1] := 5.15803E-01;
afAl[509, 0] := 5.45000E+03; afAl[509, 1] := 5.07232E-01;
afAl[510, 0] := 5.50000E+03; afAl[510, 1] := 4.98881E-01;
afAl[511, 0] := 5.55000E+03; afAl[511, 1] := 4.90742E-01;
afAl[512, 0] := 5.60000E+03; afAl[512, 1] := 4.82807E-01;
afAl[513, 0] := 5.65000E+03; afAl[513, 1] := 4.75067E-01;
afAl[514, 0] := 5.70000E+03; afAl[514, 1] := 4.67516E-01;
afAl[515, 0] := 5.75000E+03; afAl[515, 1] := 4.60153E-01;
afAl[516, 0] := 5.80000E+03; afAl[516, 1] := 4.52969E-01;
afAl[517, 0] := 5.85000E+03; afAl[517, 1] := 4.45958E-01;
afAl[518, 0] := 5.90000E+03; afAl[518, 1] := 4.39117E-01;
afAl[519, 0] := 5.95000E+03; afAl[519, 1] := 4.32433E-01;
afAl[520, 0] := 6.00000E+03; afAl[520, 1] := 4.25904E-01;
afAl[521, 0] := 6.05000E+03; afAl[521, 1] := 4.19532E-01;
afAl[522, 0] := 6.10000E+03; afAl[522, 1] := 4.13308E-01;
afAl[523, 0] := 6.15000E+03; afAl[523, 1] := 4.07223E-01;
afAl[524, 0] := 6.20000E+03; afAl[524, 1] := 4.01273E-01;
afAl[525, 0] := 6.25000E+03; afAl[525, 1] := 3.95461E-01;
afAl[526, 0] := 6.30000E+03; afAl[526, 1] := 3.89780E-01;
afAl[527, 0] := 6.35000E+03; afAl[527, 1] := 3.84221E-01;
afAl[528, 0] := 6.40000E+03; afAl[528, 1] := 3.78787E-01;
afAl[529, 0] := 6.45000E+03; afAl[529, 1] := 3.73469E-01;
afAl[530, 0] := 6.50000E+03; afAl[530, 1] := 3.68265E-01;
afAl[531, 0] := 6.55000E+03; afAl[531, 1] := 3.63172E-01;
afAl[532, 0] := 6.60000E+03; afAl[532, 1] := 3.58189E-01;
afAl[533, 0] := 6.65000E+03; afAl[533, 1] := 3.53312E-01;
afAl[534, 0] := 6.70000E+03; afAl[534, 1] := 3.48540E-01;
afAl[535, 0] := 6.75000E+03; afAl[535, 1] := 3.43831E-01;
afAl[536, 0] := 6.80000E+03; afAl[536, 1] := 3.39040E-01;
afAl[537, 0] := 6.85000E+03; afAl[537, 1] := 3.34294E-01;
afAl[538, 0] := 6.90000E+03; afAl[538, 1] := 3.29636E-01;
afAl[539, 0] := 6.95000E+03; afAl[539, 1] := 3.25075E-01;
afAl[540, 0] := 7.00000E+03; afAl[540, 1] := 3.20609E-01;
afAl[541, 0] := 7.05000E+03; afAl[541, 1] := 3.16237E-01;
afAl[542, 0] := 7.10000E+03; afAl[542, 1] := 3.11954E-01;
afAl[543, 0] := 7.15000E+03; afAl[543, 1] := 3.07756E-01;
afAl[544, 0] := 7.20000E+03; afAl[544, 1] := 3.03648E-01;
afAl[545, 0] := 7.25000E+03; afAl[545, 1] := 2.99622E-01;
afAl[546, 0] := 7.30000E+03; afAl[546, 1] := 2.95676E-01;
afAl[547, 0] := 7.35000E+03; afAl[547, 1] := 2.91802E-01;
afAl[548, 0] := 7.40000E+03; afAl[548, 1] := 2.88010E-01;
afAl[549, 0] := 7.45000E+03; afAl[549, 1] := 2.84296E-01;
afAl[550, 0] := 7.50000E+03; afAl[550, 1] := 2.80651E-01;
afAl[551, 0] := 7.55000E+03; afAl[551, 1] := 2.77076E-01;
afAl[552, 0] := 7.60000E+03; afAl[552, 1] := 2.73568E-01;
afAl[553, 0] := 7.65000E+03; afAl[553, 1] := 2.70134E-01;
afAl[554, 0] := 7.70000E+03; afAl[554, 1] := 2.66761E-01;
afAl[555, 0] := 7.75000E+03; afAl[555, 1] := 2.63449E-01;
afAl[556, 0] := 7.80000E+03; afAl[556, 1] := 2.60201E-01;
afAl[557, 0] := 7.85000E+03; afAl[557, 1] := 2.57015E-01;
afAl[558, 0] := 7.90000E+03; afAl[558, 1] := 2.53890E-01;
afAl[559, 0] := 7.95000E+03; afAl[559, 1] := 2.50820E-01;
afAl[560, 0] := 8.00000E+03; afAl[560, 1] := 2.47805E-01;
afAl[561, 0] := 8.05000E+03; afAl[561, 1] := 2.44844E-01;
afAl[562, 0] := 8.10000E+03; afAl[562, 1] := 2.41937E-01;
afAl[563, 0] := 8.15000E+03; afAl[563, 1] := 2.39082E-01;
afAl[564, 0] := 8.20000E+03; afAl[564, 1] := 2.36279E-01;
afAl[565, 0] := 8.25000E+03; afAl[565, 1] := 2.33527E-01;
afAl[566, 0] := 8.30000E+03; afAl[566, 1] := 2.30824E-01;
afAl[567, 0] := 8.35000E+03; afAl[567, 1] := 2.28165E-01;
afAl[568, 0] := 8.40000E+03; afAl[568, 1] := 2.25553E-01;
afAl[569, 0] := 8.45000E+03; afAl[569, 1] := 2.22984E-01;
afAl[570, 0] := 8.50000E+03; afAl[570, 1] := 2.20461E-01;
afAl[571, 0] := 8.55000E+03; afAl[571, 1] := 2.17984E-01;
afAl[572, 0] := 8.60000E+03; afAl[572, 1] := 2.15549E-01;
afAl[573, 0] := 8.65000E+03; afAl[573, 1] := 2.13155E-01;
afAl[574, 0] := 8.70000E+03; afAl[574, 1] := 2.10796E-01;
afAl[575, 0] := 8.75000E+03; afAl[575, 1] := 2.08477E-01;
afAl[576, 0] := 8.80000E+03; afAl[576, 1] := 2.06198E-01;
afAl[577, 0] := 8.85000E+03; afAl[577, 1] := 2.03951E-01;
afAl[578, 0] := 8.90000E+03; afAl[578, 1] := 2.01737E-01;
afAl[579, 0] := 8.95000E+03; afAl[579, 1] := 1.99445E-01;
afAl[580, 0] := 9.00000E+03; afAl[580, 1] := 1.97174E-01;
afAl[581, 0] := 9.05000E+03; afAl[581, 1] := 1.94944E-01;
afAl[582, 0] := 9.10000E+03; afAl[582, 1] := 1.92750E-01;
afAl[583, 0] := 9.15000E+03; afAl[583, 1] := 1.90588E-01;
afAl[584, 0] := 9.20000E+03; afAl[584, 1] := 1.88465E-01;
afAl[585, 0] := 9.25000E+03; afAl[585, 1] := 1.86380E-01;
afAl[586, 0] := 9.30000E+03; afAl[586, 1] := 1.84326E-01;
afAl[587, 0] := 9.35000E+03; afAl[587, 1] := 1.82305E-01;
afAl[588, 0] := 9.40000E+03; afAl[588, 1] := 1.80317E-01;
afAl[589, 0] := 9.45000E+03; afAl[589, 1] := 1.78363E-01;
afAl[590, 0] := 9.50000E+03; afAl[590, 1] := 1.76437E-01;
afAl[591, 0] := 9.55000E+03; afAl[591, 1] := 1.74542E-01;
afAl[592, 0] := 9.60000E+03; afAl[592, 1] := 1.72675E-01;
afAl[593, 0] := 9.65000E+03; afAl[593, 1] := 1.70839E-01;
afAl[594, 0] := 9.70000E+03; afAl[594, 1] := 1.69035E-01;
afAl[595, 0] := 9.75000E+03; afAl[595, 1] := 1.67259E-01;
afAl[596, 0] := 9.80000E+03; afAl[596, 1] := 1.65511E-01;
afAl[597, 0] := 9.85000E+03; afAl[597, 1] := 1.63790E-01;
afAl[598, 0] := 9.90000E+03; afAl[598, 1] := 1.62096E-01;
afAl[599, 0] := 9.95000E+03; afAl[599, 1] := 1.60427E-01;
afAl[600, 0] := 1.00000E+04; afAl[600, 1] := 1.58780E-01;
afAl[601, 0] := 1.00500E+04; afAl[601, 1] := 1.57160E-01;
afAl[602, 0] := 1.01000E+04; afAl[602, 1] := 1.55565E-01;
afAl[603, 0] := 1.01500E+04; afAl[603, 1] := 1.53993E-01;
afAl[604, 0] := 1.02000E+04; afAl[604, 1] := 1.52444E-01;
afAl[605, 0] := 1.02500E+04; afAl[605, 1] := 1.50918E-01;
afAl[606, 0] := 1.03000E+04; afAl[606, 1] := 1.49417E-01;
afAl[607, 0] := 1.03500E+04; afAl[607, 1] := 1.47938E-01;
afAl[608, 0] := 1.04000E+04; afAl[608, 1] := 1.46480E-01;
afAl[609, 0] := 1.04500E+04; afAl[609, 1] := 1.45043E-01;
afAl[610, 0] := 1.05000E+04; afAl[610, 1] := 1.43627E-01;
afAl[611, 0] := 1.05500E+04; afAl[611, 1] := 1.42231E-01;
afAl[612, 0] := 1.06000E+04; afAl[612, 1] := 1.40856E-01;
afAl[613, 0] := 1.06500E+04; afAl[613, 1] := 1.39500E-01;
afAl[614, 0] := 1.07000E+04; afAl[614, 1] := 1.38164E-01;
afAl[615, 0] := 1.07500E+04; afAl[615, 1] := 1.36848E-01;
afAl[616, 0] := 1.08000E+04; afAl[616, 1] := 1.35551E-01;
afAl[617, 0] := 1.08500E+04; afAl[617, 1] := 1.34272E-01;
afAl[618, 0] := 1.09000E+04; afAl[618, 1] := 1.33010E-01;
afAl[619, 0] := 1.09500E+04; afAl[619, 1] := 1.31764E-01;
afAl[620, 0] := 1.10000E+04; afAl[620, 1] := 1.30536E-01;
afAl[621, 0] := 1.10500E+04; afAl[621, 1] := 1.29327E-01;
afAl[622, 0] := 1.11000E+04; afAl[622, 1] := 1.28134E-01;
afAl[623, 0] := 1.11500E+04; afAl[623, 1] := 1.26956E-01;
afAl[624, 0] := 1.12000E+04; afAl[624, 1] := 1.25794E-01;
afAl[625, 0] := 1.12500E+04; afAl[625, 1] := 1.24646E-01;
afAl[626, 0] := 1.13000E+04; afAl[626, 1] := 1.23514E-01;
afAl[627, 0] := 1.13500E+04; afAl[627, 1] := 1.22397E-01;
afAl[628, 0] := 1.14000E+04; afAl[628, 1] := 1.21294E-01;
afAl[629, 0] := 1.14500E+04; afAl[629, 1] := 1.20209E-01;
afAl[630, 0] := 1.15000E+04; afAl[630, 1] := 1.19139E-01;
afAl[631, 0] := 1.15500E+04; afAl[631, 1] := 1.18083E-01;
afAl[632, 0] := 1.16000E+04; afAl[632, 1] := 1.17037E-01;
afAl[633, 0] := 1.16500E+04; afAl[633, 1] := 1.16006E-01;
afAl[634, 0] := 1.17000E+04; afAl[634, 1] := 1.14992E-01;
afAl[635, 0] := 1.17500E+04; afAl[635, 1] := 1.13992E-01;
afAl[636, 0] := 1.18000E+04; afAl[636, 1] := 1.13002E-01;
afAl[637, 0] := 1.18500E+04; afAl[637, 1] := 1.12025E-01;
afAl[638, 0] := 1.19000E+04; afAl[638, 1] := 1.11060E-01;
afAl[639, 0] := 1.19500E+04; afAl[639, 1] := 1.10108E-01;
afAl[640, 0] := 1.20000E+04; afAl[640, 1] := 1.09169E-01;
afAl[641, 0] := 1.20500E+04; afAl[641, 1] := 1.08239E-01;
afAl[642, 0] := 1.21000E+04; afAl[642, 1] := 1.07321E-01;
afAl[643, 0] := 1.21500E+04; afAl[643, 1] := 1.06416E-01;
afAl[644, 0] := 1.22000E+04; afAl[644, 1] := 1.05522E-01;
afAl[645, 0] := 1.22500E+04; afAl[645, 1] := 1.04640E-01;
afAl[646, 0] := 1.23000E+04; afAl[646, 1] := 1.03768E-01;
afAl[647, 0] := 1.23500E+04; afAl[647, 1] := 1.02906E-01;
afAl[648, 0] := 1.24000E+04; afAl[648, 1] := 1.02054E-01;
afAl[649, 0] := 1.24500E+04; afAl[649, 1] := 1.01212E-01;
afAl[650, 0] := 1.25000E+04; afAl[650, 1] := 1.00381E-01;
afAl[651, 0] := 1.25500E+04; afAl[651, 1] := 9.95618E-02;
afAl[652, 0] := 1.26000E+04; afAl[652, 1] := 9.87529E-02;
afAl[653, 0] := 1.26500E+04; afAl[653, 1] := 9.79529E-02;
afAl[654, 0] := 1.27000E+04; afAl[654, 1] := 9.71620E-02;
afAl[655, 0] := 1.27500E+04; afAl[655, 1] := 9.63807E-02;
afAl[656, 0] := 1.28000E+04; afAl[656, 1] := 9.56089E-02;
afAl[657, 0] := 1.28500E+04; afAl[657, 1] := 9.48462E-02;
afAl[658, 0] := 1.29000E+04; afAl[658, 1] := 9.40927E-02;
afAl[659, 0] := 1.29500E+04; afAl[659, 1] := 9.33481E-02;
afAl[660, 0] := 1.30000E+04; afAl[660, 1] := 9.26123E-02;
afAl[661, 0] := 1.30500E+04; afAl[661, 1] := 9.18847E-02;
afAl[662, 0] := 1.31000E+04; afAl[662, 1] := 9.11657E-02;
afAl[663, 0] := 1.31500E+04; afAl[663, 1] := 9.04550E-02;
afAl[664, 0] := 1.32000E+04; afAl[664, 1] := 8.97525E-02;
afAl[665, 0] := 1.32500E+04; afAl[665, 1] := 8.90581E-02;
afAl[666, 0] := 1.33000E+04; afAl[666, 1] := 8.83719E-02;
afAl[667, 0] := 1.33500E+04; afAl[667, 1] := 8.76936E-02;
afAl[668, 0] := 1.34000E+04; afAl[668, 1] := 8.70229E-02;
afAl[669, 0] := 1.34500E+04; afAl[669, 1] := 8.63595E-02;
afAl[670, 0] := 1.35000E+04; afAl[670, 1] := 8.57034E-02;
afAl[671, 0] := 1.35500E+04; afAl[671, 1] := 8.50550E-02;
afAl[672, 0] := 1.36000E+04; afAl[672, 1] := 8.44142E-02;
afAl[673, 0] := 1.36500E+04; afAl[673, 1] := 8.37805E-02;
afAl[674, 0] := 1.37000E+04; afAl[674, 1] := 8.31536E-02;
afAl[675, 0] := 1.37500E+04; afAl[675, 1] := 8.25335E-02;
afAl[676, 0] := 1.38000E+04; afAl[676, 1] := 8.19203E-02;
afAl[677, 0] := 1.38500E+04; afAl[677, 1] := 8.13141E-02;
afAl[678, 0] := 1.39000E+04; afAl[678, 1] := 8.07146E-02;
afAl[679, 0] := 1.39500E+04; afAl[679, 1] := 8.01216E-02;
afAl[680, 0] := 1.40000E+04; afAl[680, 1] := 7.95349E-02;
afAl[681, 0] := 1.40500E+04; afAl[681, 1] := 7.89546E-02;
afAl[682, 0] := 1.41000E+04; afAl[682, 1] := 7.83805E-02;
afAl[683, 0] := 1.41500E+04; afAl[683, 1] := 7.78127E-02;
afAl[684, 0] := 1.42000E+04; afAl[684, 1] := 7.72509E-02;
afAl[685, 0] := 1.42500E+04; afAl[685, 1] := 7.66954E-02;
afAl[686, 0] := 1.43000E+04; afAl[686, 1] := 7.61459E-02;
afAl[687, 0] := 1.43500E+04; afAl[687, 1] := 7.56022E-02;
afAl[688, 0] := 1.44000E+04; afAl[688, 1] := 7.50641E-02;
afAl[689, 0] := 1.44500E+04; afAl[689, 1] := 7.45317E-02;
afAl[690, 0] := 1.45000E+04; afAl[690, 1] := 7.40048E-02;
afAl[691, 0] := 1.45500E+04; afAl[691, 1] := 7.34836E-02;
afAl[692, 0] := 1.46000E+04; afAl[692, 1] := 7.29677E-02;
afAl[693, 0] := 1.46500E+04; afAl[693, 1] := 7.24572E-02;
afAl[694, 0] := 1.47000E+04; afAl[694, 1] := 7.19520E-02;
afAl[695, 0] := 1.47500E+04; afAl[695, 1] := 7.14519E-02;
afAl[696, 0] := 1.48000E+04; afAl[696, 1] := 7.09570E-02;
afAl[697, 0] := 1.48500E+04; afAl[697, 1] := 7.04670E-02;
afAl[698, 0] := 1.49000E+04; afAl[698, 1] := 6.99819E-02;
afAl[699, 0] := 1.49500E+04; afAl[699, 1] := 6.95019E-02;
afAl[700, 0] := 1.50000E+04; afAl[700, 1] := 6.90270E-02;
afAl[701, 0] := 1.50500E+04; afAl[701, 1] := 6.85569E-02;
afAl[702, 0] := 1.51000E+04; afAl[702, 1] := 6.80916E-02;
afAl[703, 0] := 1.51500E+04; afAl[703, 1] := 6.76311E-02;
afAl[704, 0] := 1.52000E+04; afAl[704, 1] := 6.71753E-02;
afAl[705, 0] := 1.52500E+04; afAl[705, 1] := 6.67239E-02;
afAl[706, 0] := 1.53000E+04; afAl[706, 1] := 6.62768E-02;
afAl[707, 0] := 1.53500E+04; afAl[707, 1] := 6.58342E-02;
afAl[708, 0] := 1.54000E+04; afAl[708, 1] := 6.53959E-02;
afAl[709, 0] := 1.54500E+04; afAl[709, 1] := 6.49618E-02;
afAl[710, 0] := 1.55000E+04; afAl[710, 1] := 6.45320E-02;
afAl[711, 0] := 1.55500E+04; afAl[711, 1] := 6.41065E-02;
afAl[712, 0] := 1.56000E+04; afAl[712, 1] := 6.36854E-02;
afAl[713, 0] := 1.56500E+04; afAl[713, 1] := 6.32685E-02;
afAl[714, 0] := 1.57000E+04; afAl[714, 1] := 6.28556E-02;
afAl[715, 0] := 1.57500E+04; afAl[715, 1] := 6.24464E-02;
afAl[716, 0] := 1.58000E+04; afAl[716, 1] := 6.20411E-02;
afAl[717, 0] := 1.58500E+04; afAl[717, 1] := 6.16397E-02;
afAl[718, 0] := 1.59000E+04; afAl[718, 1] := 6.12424E-02;
afAl[719, 0] := 1.59500E+04; afAl[719, 1] := 6.08490E-02;
afAl[720, 0] := 1.60000E+04; afAl[720, 1] := 6.04594E-02;
afAl[721, 0] := 1.60500E+04; afAl[721, 1] := 6.00733E-02;
afAl[722, 0] := 1.61000E+04; afAl[722, 1] := 5.96907E-02;
afAl[723, 0] := 1.61500E+04; afAl[723, 1] := 5.93116E-02;
afAl[724, 0] := 1.62000E+04; afAl[724, 1] := 5.89363E-02;
afAl[725, 0] := 1.62500E+04; afAl[725, 1] := 5.85648E-02;
afAl[726, 0] := 1.63000E+04; afAl[726, 1] := 5.81968E-02;
afAl[727, 0] := 1.63500E+04; afAl[727, 1] := 5.78321E-02;
afAl[728, 0] := 1.64000E+04; afAl[728, 1] := 5.74705E-02;
afAl[729, 0] := 1.64500E+04; afAl[729, 1] := 5.71123E-02;
afAl[730, 0] := 1.65000E+04; afAl[730, 1] := 5.67574E-02;
afAl[731, 0] := 1.65500E+04; afAl[731, 1] := 5.64058E-02;
afAl[732, 0] := 1.66000E+04; afAl[732, 1] := 5.60575E-02;
afAl[733, 0] := 1.66500E+04; afAl[733, 1] := 5.57124E-02;
afAl[734, 0] := 1.67000E+04; afAl[734, 1] := 5.53703E-02;
afAl[735, 0] := 1.67500E+04; afAl[735, 1] := 5.50314E-02;
afAl[736, 0] := 1.68000E+04; afAl[736, 1] := 5.46955E-02;
afAl[737, 0] := 1.68500E+04; afAl[737, 1] := 5.43627E-02;
afAl[738, 0] := 1.69000E+04; afAl[738, 1] := 5.40330E-02;
afAl[739, 0] := 1.69500E+04; afAl[739, 1] := 5.37062E-02;
afAl[740, 0] := 1.70000E+04; afAl[740, 1] := 5.33824E-02;
afAl[741, 0] := 1.70500E+04; afAl[741, 1] := 5.30616E-02;
afAl[742, 0] := 1.71000E+04; afAl[742, 1] := 5.27438E-02;
afAl[743, 0] := 1.71500E+04; afAl[743, 1] := 5.24287E-02;
afAl[744, 0] := 1.72000E+04; afAl[744, 1] := 5.21164E-02;
afAl[745, 0] := 1.72500E+04; afAl[745, 1] := 5.18066E-02;
afAl[746, 0] := 1.73000E+04; afAl[746, 1] := 5.14996E-02;
afAl[747, 0] := 1.73500E+04; afAl[747, 1] := 5.11953E-02;
afAl[748, 0] := 1.74000E+04; afAl[748, 1] := 5.08936E-02;
afAl[749, 0] := 1.74500E+04; afAl[749, 1] := 5.05945E-02;
afAl[750, 0] := 1.75000E+04; afAl[750, 1] := 5.02980E-02;
afAl[751, 0] := 1.75500E+04; afAl[751, 1] := 5.00042E-02;
afAl[752, 0] := 1.76000E+04; afAl[752, 1] := 4.97131E-02;
afAl[753, 0] := 1.76500E+04; afAl[753, 1] := 4.94246E-02;
afAl[754, 0] := 1.77000E+04; afAl[754, 1] := 4.91385E-02;
afAl[755, 0] := 1.77500E+04; afAl[755, 1] := 4.88547E-02;
afAl[756, 0] := 1.78000E+04; afAl[756, 1] := 4.85734E-02;
afAl[757, 0] := 1.78500E+04; afAl[757, 1] := 4.82944E-02;
afAl[758, 0] := 1.79000E+04; afAl[758, 1] := 4.80178E-02;
afAl[759, 0] := 1.79500E+04; afAl[759, 1] := 4.77436E-02;
afAl[760, 0] := 1.80000E+04; afAl[760, 1] := 4.74717E-02;
afAl[761, 0] := 1.80500E+04; afAl[761, 1] := 4.72021E-02;
afAl[762, 0] := 1.81000E+04; afAl[762, 1] := 4.69348E-02;
afAl[763, 0] := 1.81500E+04; afAl[763, 1] := 4.66698E-02;
afAl[764, 0] := 1.82000E+04; afAl[764, 1] := 4.64070E-02;
afAl[765, 0] := 1.82500E+04; afAl[765, 1] := 4.61463E-02;
afAl[766, 0] := 1.83000E+04; afAl[766, 1] := 4.58878E-02;
afAl[767, 0] := 1.83500E+04; afAl[767, 1] := 4.56314E-02;
afAl[768, 0] := 1.84000E+04; afAl[768, 1] := 4.53772E-02;
afAl[769, 0] := 1.84500E+04; afAl[769, 1] := 4.51251E-02;
afAl[770, 0] := 1.85000E+04; afAl[770, 1] := 4.48750E-02;
afAl[771, 0] := 1.85500E+04; afAl[771, 1] := 4.46270E-02;
afAl[772, 0] := 1.86000E+04; afAl[772, 1] := 4.43811E-02;
afAl[773, 0] := 1.86500E+04; afAl[773, 1] := 4.41373E-02;
afAl[774, 0] := 1.87000E+04; afAl[774, 1] := 4.38954E-02;
afAl[775, 0] := 1.87500E+04; afAl[775, 1] := 4.36556E-02;
afAl[776, 0] := 1.88000E+04; afAl[776, 1] := 4.34176E-02;
afAl[777, 0] := 1.88500E+04; afAl[777, 1] := 4.31816E-02;
afAl[778, 0] := 1.89000E+04; afAl[778, 1] := 4.29475E-02;
afAl[779, 0] := 1.89500E+04; afAl[779, 1] := 4.27152E-02;
afAl[780, 0] := 1.90000E+04; afAl[780, 1] := 4.24847E-02;
afAl[781, 0] := 1.90500E+04; afAl[781, 1] := 4.22560E-02;
afAl[782, 0] := 1.91000E+04; afAl[782, 1] := 4.20291E-02;
afAl[783, 0] := 1.91500E+04; afAl[783, 1] := 4.18040E-02;
afAl[784, 0] := 1.92000E+04; afAl[784, 1] := 4.15808E-02;
afAl[785, 0] := 1.92500E+04; afAl[785, 1] := 4.13594E-02;
afAl[786, 0] := 1.93000E+04; afAl[786, 1] := 4.11397E-02;
afAl[787, 0] := 1.93500E+04; afAl[787, 1] := 4.09218E-02;
afAl[788, 0] := 1.94000E+04; afAl[788, 1] := 4.07055E-02;
afAl[789, 0] := 1.94500E+04; afAl[789, 1] := 4.04910E-02;
afAl[790, 0] := 1.95000E+04; afAl[790, 1] := 4.02782E-02;
afAl[791, 0] := 1.95500E+04; afAl[791, 1] := 4.00670E-02;
afAl[792, 0] := 1.96000E+04; afAl[792, 1] := 3.98575E-02;
afAl[793, 0] := 1.96500E+04; afAl[793, 1] := 3.96496E-02;
afAl[794, 0] := 1.97000E+04; afAl[794, 1] := 3.94434E-02;
afAl[795, 0] := 1.97500E+04; afAl[795, 1] := 3.92387E-02;
afAl[796, 0] := 1.98000E+04; afAl[796, 1] := 3.90355E-02;
afAl[797, 0] := 1.98500E+04; afAl[797, 1] := 3.88339E-02;
afAl[798, 0] := 1.99000E+04; afAl[798, 1] := 3.86338E-02;
afAl[799, 0] := 1.99500E+04; afAl[799, 1] := 3.84353E-02;
afAl[800, 0] := 2.00000E+04; afAl[800, 1] := 3.82382E-02;
afAl[801, 0] := 2.00500E+04; afAl[801, 1] := 3.80427E-02;
afAl[802, 0] := 2.01000E+04; afAl[802, 1] := 3.78486E-02;
afAl[803, 0] := 2.01500E+04; afAl[803, 1] := 3.76560E-02;
afAl[804, 0] := 2.02000E+04; afAl[804, 1] := 3.74649E-02;
afAl[805, 0] := 2.02500E+04; afAl[805, 1] := 3.72753E-02;
afAl[806, 0] := 2.03000E+04; afAl[806, 1] := 3.70871E-02;
afAl[807, 0] := 2.03500E+04; afAl[807, 1] := 3.69003E-02;
afAl[808, 0] := 2.04000E+04; afAl[808, 1] := 3.67151E-02;
afAl[809, 0] := 2.04500E+04; afAl[809, 1] := 3.65312E-02;
afAl[810, 0] := 2.05000E+04; afAl[810, 1] := 3.63487E-02;
afAl[811, 0] := 2.05500E+04; afAl[811, 1] := 3.61675E-02;
afAl[812, 0] := 2.06000E+04; afAl[812, 1] := 3.59874E-02;
afAl[813, 0] := 2.06500E+04; afAl[813, 1] := 3.58086E-02;
afAl[814, 0] := 2.07000E+04; afAl[814, 1] := 3.56312E-02;
afAl[815, 0] := 2.07500E+04; afAl[815, 1] := 3.54551E-02;
afAl[816, 0] := 2.08000E+04; afAl[816, 1] := 3.52805E-02;
afAl[817, 0] := 2.08500E+04; afAl[817, 1] := 3.51072E-02;
afAl[818, 0] := 2.09000E+04; afAl[818, 1] := 3.49352E-02;
afAl[819, 0] := 2.09500E+04; afAl[819, 1] := 3.47645E-02;
afAl[820, 0] := 2.10000E+04; afAl[820, 1] := 3.45947E-02;
afAl[821, 0] := 2.10500E+04; afAl[821, 1] := 3.44260E-02;
afAl[822, 0] := 2.11000E+04; afAl[822, 1] := 3.42586E-02;
afAl[823, 0] := 2.11500E+04; afAl[823, 1] := 3.40924E-02;
afAl[824, 0] := 2.12000E+04; afAl[824, 1] := 3.39274E-02;
afAl[825, 0] := 2.12500E+04; afAl[825, 1] := 3.37638E-02;
afAl[826, 0] := 2.13000E+04; afAl[826, 1] := 3.36013E-02;
afAl[827, 0] := 2.13500E+04; afAl[827, 1] := 3.34400E-02;
afAl[828, 0] := 2.14000E+04; afAl[828, 1] := 3.32798E-02;
afAl[829, 0] := 2.14500E+04; afAl[829, 1] := 3.31208E-02;
afAl[830, 0] := 2.15000E+04; afAl[830, 1] := 3.29629E-02;
afAl[831, 0] := 2.15500E+04; afAl[831, 1] := 3.28062E-02;
afAl[832, 0] := 2.16000E+04; afAl[832, 1] := 3.26505E-02;
afAl[833, 0] := 2.16500E+04; afAl[833, 1] := 3.24960E-02;
afAl[834, 0] := 2.17000E+04; afAl[834, 1] := 3.23426E-02;
afAl[835, 0] := 2.17500E+04; afAl[835, 1] := 3.21903E-02;
afAl[836, 0] := 2.18000E+04; afAl[836, 1] := 3.20391E-02;
afAl[837, 0] := 2.18500E+04; afAl[837, 1] := 3.18888E-02;
afAl[838, 0] := 2.19000E+04; afAl[838, 1] := 3.17396E-02;
afAl[839, 0] := 2.19500E+04; afAl[839, 1] := 3.15914E-02;
afAl[840, 0] := 2.20000E+04; afAl[840, 1] := 3.14442E-02;
afAl[841, 0] := 2.20500E+04; afAl[841, 1] := 3.12980E-02;
afAl[842, 0] := 2.21000E+04; afAl[842, 1] := 3.11529E-02;
afAl[843, 0] := 2.21500E+04; afAl[843, 1] := 3.10087E-02;
afAl[844, 0] := 2.22000E+04; afAl[844, 1] := 3.08655E-02;
afAl[845, 0] := 2.22500E+04; afAl[845, 1] := 3.07233E-02;
afAl[846, 0] := 2.23000E+04; afAl[846, 1] := 3.05822E-02;
afAl[847, 0] := 2.23500E+04; afAl[847, 1] := 3.04419E-02;
afAl[848, 0] := 2.24000E+04; afAl[848, 1] := 3.03027E-02;
afAl[849, 0] := 2.24500E+04; afAl[849, 1] := 3.01644E-02;
afAl[850, 0] := 2.25000E+04; afAl[850, 1] := 3.00269E-02;
afAl[851, 0] := 2.25500E+04; afAl[851, 1] := 2.98903E-02;
afAl[852, 0] := 2.26000E+04; afAl[852, 1] := 2.97547E-02;
afAl[853, 0] := 2.26500E+04; afAl[853, 1] := 2.96200E-02;
afAl[854, 0] := 2.27000E+04; afAl[854, 1] := 2.94861E-02;
afAl[855, 0] := 2.27500E+04; afAl[855, 1] := 2.93533E-02;
afAl[856, 0] := 2.28000E+04; afAl[856, 1] := 2.92215E-02;
afAl[857, 0] := 2.28500E+04; afAl[857, 1] := 2.90904E-02;
afAl[858, 0] := 2.29000E+04; afAl[858, 1] := 2.89603E-02;
afAl[859, 0] := 2.29500E+04; afAl[859, 1] := 2.88310E-02;
afAl[860, 0] := 2.30000E+04; afAl[860, 1] := 2.87026E-02;
afAl[861, 0] := 2.30500E+04; afAl[861, 1] := 2.85750E-02;
afAl[862, 0] := 2.31000E+04; afAl[862, 1] := 2.84482E-02;
afAl[863, 0] := 2.31500E+04; afAl[863, 1] := 2.83223E-02;
afAl[864, 0] := 2.32000E+04; afAl[864, 1] := 2.81971E-02;
afAl[865, 0] := 2.32500E+04; afAl[865, 1] := 2.80726E-02;
afAl[866, 0] := 2.33000E+04; afAl[866, 1] := 2.79490E-02;
afAl[867, 0] := 2.33500E+04; afAl[867, 1] := 2.78262E-02;
afAl[868, 0] := 2.34000E+04; afAl[868, 1] := 2.77042E-02;
afAl[869, 0] := 2.34500E+04; afAl[869, 1] := 2.75831E-02;
afAl[870, 0] := 2.35000E+04; afAl[870, 1] := 2.74628E-02;
afAl[871, 0] := 2.35500E+04; afAl[871, 1] := 2.73432E-02;
afAl[872, 0] := 2.36000E+04; afAl[872, 1] := 2.72244E-02;
afAl[873, 0] := 2.36500E+04; afAl[873, 1] := 2.71065E-02;
afAl[874, 0] := 2.37000E+04; afAl[874, 1] := 2.69893E-02;
afAl[875, 0] := 2.37500E+04; afAl[875, 1] := 2.68730E-02;
afAl[876, 0] := 2.38000E+04; afAl[876, 1] := 2.67573E-02;
afAl[877, 0] := 2.38500E+04; afAl[877, 1] := 2.66424E-02;
afAl[878, 0] := 2.39000E+04; afAl[878, 1] := 2.65281E-02;
afAl[879, 0] := 2.39500E+04; afAl[879, 1] := 2.64144E-02;
afAl[880, 0] := 2.40000E+04; afAl[880, 1] := 2.63015E-02;
afAl[881, 0] := 2.40500E+04; afAl[881, 1] := 2.61892E-02;
afAl[882, 0] := 2.41000E+04; afAl[882, 1] := 2.60778E-02;
afAl[883, 0] := 2.41500E+04; afAl[883, 1] := 2.59672E-02;
afAl[884, 0] := 2.42000E+04; afAl[884, 1] := 2.58573E-02;
afAl[885, 0] := 2.42500E+04; afAl[885, 1] := 2.57481E-02;
afAl[886, 0] := 2.43000E+04; afAl[886, 1] := 2.56396E-02;
afAl[887, 0] := 2.43500E+04; afAl[887, 1] := 2.55317E-02;
afAl[888, 0] := 2.44000E+04; afAl[888, 1] := 2.54244E-02;
afAl[889, 0] := 2.44500E+04; afAl[889, 1] := 2.53178E-02;
afAl[890, 0] := 2.45000E+04; afAl[890, 1] := 2.52118E-02;
afAl[891, 0] := 2.45500E+04; afAl[891, 1] := 2.51065E-02;
afAl[892, 0] := 2.46000E+04; afAl[892, 1] := 2.50020E-02;
afAl[893, 0] := 2.46500E+04; afAl[893, 1] := 2.48981E-02;
afAl[894, 0] := 2.47000E+04; afAl[894, 1] := 2.47948E-02;
afAl[895, 0] := 2.47500E+04; afAl[895, 1] := 2.46922E-02;
afAl[896, 0] := 2.48000E+04; afAl[896, 1] := 2.45902E-02;
afAl[897, 0] := 2.48500E+04; afAl[897, 1] := 2.44889E-02;
afAl[898, 0] := 2.49000E+04; afAl[898, 1] := 2.43881E-02;
afAl[899, 0] := 2.49500E+04; afAl[899, 1] := 2.42879E-02;
afAl[900, 0] := 2.50000E+04; afAl[900, 1] := 2.41884E-02;
afAl[901, 0] := 2.50500E+04; afAl[901, 1] := 2.40894E-02;
afAl[902, 0] := 2.51000E+04; afAl[902, 1] := 2.39909E-02;
afAl[903, 0] := 2.51500E+04; afAl[903, 1] := 2.38930E-02;
afAl[904, 0] := 2.52000E+04; afAl[904, 1] := 2.37956E-02;
afAl[905, 0] := 2.52500E+04; afAl[905, 1] := 2.36988E-02;
afAl[906, 0] := 2.53000E+04; afAl[906, 1] := 2.36027E-02;
afAl[907, 0] := 2.53500E+04; afAl[907, 1] := 2.35072E-02;
afAl[908, 0] := 2.54000E+04; afAl[908, 1] := 2.34124E-02;
afAl[909, 0] := 2.54500E+04; afAl[909, 1] := 2.33181E-02;
afAl[910, 0] := 2.55000E+04; afAl[910, 1] := 2.32244E-02;
afAl[911, 0] := 2.55500E+04; afAl[911, 1] := 2.31313E-02;
afAl[912, 0] := 2.56000E+04; afAl[912, 1] := 2.30388E-02;
afAl[913, 0] := 2.56500E+04; afAl[913, 1] := 2.29469E-02;
afAl[914, 0] := 2.57000E+04; afAl[914, 1] := 2.28555E-02;
afAl[915, 0] := 2.57500E+04; afAl[915, 1] := 2.27646E-02;
afAl[916, 0] := 2.58000E+04; afAl[916, 1] := 2.26743E-02;
afAl[917, 0] := 2.58500E+04; afAl[917, 1] := 2.25844E-02;
afAl[918, 0] := 2.59000E+04; afAl[918, 1] := 2.24949E-02;
afAl[919, 0] := 2.59500E+04; afAl[919, 1] := 2.24059E-02;
afAl[920, 0] := 2.60000E+04; afAl[920, 1] := 2.23174E-02;
afAl[921, 0] := 2.60500E+04; afAl[921, 1] := 2.22294E-02;
afAl[922, 0] := 2.61000E+04; afAl[922, 1] := 2.21420E-02;
afAl[923, 0] := 2.61500E+04; afAl[923, 1] := 2.20552E-02;
afAl[924, 0] := 2.62000E+04; afAl[924, 1] := 2.19689E-02;
afAl[925, 0] := 2.62500E+04; afAl[925, 1] := 2.18831E-02;
afAl[926, 0] := 2.63000E+04; afAl[926, 1] := 2.17978E-02;
afAl[927, 0] := 2.63500E+04; afAl[927, 1] := 2.17130E-02;
afAl[928, 0] := 2.64000E+04; afAl[928, 1] := 2.16289E-02;
afAl[929, 0] := 2.64500E+04; afAl[929, 1] := 2.15452E-02;
afAl[930, 0] := 2.65000E+04; afAl[930, 1] := 2.14621E-02;
afAl[931, 0] := 2.65500E+04; afAl[931, 1] := 2.13794E-02;
afAl[932, 0] := 2.66000E+04; afAl[932, 1] := 2.12972E-02;
afAl[933, 0] := 2.66500E+04; afAl[933, 1] := 2.12134E-02;
afAl[934, 0] := 2.67000E+04; afAl[934, 1] := 2.11295E-02;
afAl[935, 0] := 2.67500E+04; afAl[935, 1] := 2.10461E-02;
afAl[936, 0] := 2.68000E+04; afAl[936, 1] := 2.09631E-02;
afAl[937, 0] := 2.68500E+04; afAl[937, 1] := 2.08807E-02;
afAl[938, 0] := 2.69000E+04; afAl[938, 1] := 2.07983E-02;
afAl[939, 0] := 2.69500E+04; afAl[939, 1] := 2.07158E-02;
afAl[940, 0] := 2.70000E+04; afAl[940, 1] := 2.06337E-02;
afAl[941, 0] := 2.70500E+04; afAl[941, 1] := 2.05522E-02;
afAl[942, 0] := 2.71000E+04; afAl[942, 1] := 2.04711E-02;
afAl[943, 0] := 2.71500E+04; afAl[943, 1] := 2.03905E-02;
afAl[944, 0] := 2.72000E+04; afAl[944, 1] := 2.03105E-02;
afAl[945, 0] := 2.72500E+04; afAl[945, 1] := 2.02310E-02;
afAl[946, 0] := 2.73000E+04; afAl[946, 1] := 2.01519E-02;
afAl[947, 0] := 2.73500E+04; afAl[947, 1] := 2.00733E-02;
afAl[948, 0] := 2.74000E+04; afAl[948, 1] := 1.99951E-02;
afAl[949, 0] := 2.74500E+04; afAl[949, 1] := 1.99173E-02;
afAl[950, 0] := 2.75000E+04; afAl[950, 1] := 1.98398E-02;
afAl[951, 0] := 2.75500E+04; afAl[951, 1] := 1.97627E-02;
afAl[952, 0] := 2.76000E+04; afAl[952, 1] := 1.96861E-02;
afAl[953, 0] := 2.76500E+04; afAl[953, 1] := 1.96100E-02;
afAl[954, 0] := 2.77000E+04; afAl[954, 1] := 1.95342E-02;
afAl[955, 0] := 2.77500E+04; afAl[955, 1] := 1.94590E-02;
afAl[956, 0] := 2.78000E+04; afAl[956, 1] := 1.93841E-02;
afAl[957, 0] := 2.78500E+04; afAl[957, 1] := 1.93097E-02;
afAl[958, 0] := 2.79000E+04; afAl[958, 1] := 1.92356E-02;
afAl[959, 0] := 2.79500E+04; afAl[959, 1] := 1.91620E-02;
afAl[960, 0] := 2.80000E+04; afAl[960, 1] := 1.90889E-02;
afAl[961, 0] := 2.80500E+04; afAl[961, 1] := 1.90162E-02;
afAl[962, 0] := 2.81000E+04; afAl[962, 1] := 1.89438E-02;
afAl[963, 0] := 2.81500E+04; afAl[963, 1] := 1.88719E-02;
afAl[964, 0] := 2.82000E+04; afAl[964, 1] := 1.88004E-02;
afAl[965, 0] := 2.82500E+04; afAl[965, 1] := 1.87293E-02;
afAl[966, 0] := 2.83000E+04; afAl[966, 1] := 1.86587E-02;
afAl[967, 0] := 2.83500E+04; afAl[967, 1] := 1.85884E-02;
afAl[968, 0] := 2.84000E+04; afAl[968, 1] := 1.85186E-02;
afAl[969, 0] := 2.84500E+04; afAl[969, 1] := 1.84491E-02;
afAl[970, 0] := 2.85000E+04; afAl[970, 1] := 1.83800E-02;
afAl[971, 0] := 2.85500E+04; afAl[971, 1] := 1.83113E-02;
afAl[972, 0] := 2.86000E+04; afAl[972, 1] := 1.82429E-02;
afAl[973, 0] := 2.86500E+04; afAl[973, 1] := 1.81749E-02;
afAl[974, 0] := 2.87000E+04; afAl[974, 1] := 1.81073E-02;
afAl[975, 0] := 2.87500E+04; afAl[975, 1] := 1.80400E-02;
afAl[976, 0] := 2.88000E+04; afAl[976, 1] := 1.79731E-02;
afAl[977, 0] := 2.88500E+04; afAl[977, 1] := 1.79064E-02;
afAl[978, 0] := 2.89000E+04; afAl[978, 1] := 1.78400E-02;
afAl[979, 0] := 2.89500E+04; afAl[979, 1] := 1.77740E-02;
afAl[980, 0] := 2.90000E+04; afAl[980, 1] := 1.77084E-02;
afAl[981, 0] := 2.90500E+04; afAl[981, 1] := 1.76431E-02;
afAl[982, 0] := 2.91000E+04; afAl[982, 1] := 1.75781E-02;
afAl[983, 0] := 2.91500E+04; afAl[983, 1] := 1.75137E-02;
afAl[984, 0] := 2.92000E+04; afAl[984, 1] := 1.74496E-02;
afAl[985, 0] := 2.92500E+04; afAl[985, 1] := 1.73858E-02;
afAl[986, 0] := 2.93000E+04; afAl[986, 1] := 1.73225E-02;
afAl[987, 0] := 2.93500E+04; afAl[987, 1] := 1.72594E-02;
afAl[988, 0] := 2.94000E+04; afAl[988, 1] := 1.71967E-02;
afAl[989, 0] := 2.94500E+04; afAl[989, 1] := 1.71343E-02;
afAl[990, 0] := 2.95000E+04; afAl[990, 1] := 1.70723E-02;
afAl[991, 0] := 2.95500E+04; afAl[991, 1] := 1.70106E-02;
afAl[992, 0] := 2.96000E+04; afAl[992, 1] := 1.69493E-02;
afAl[993, 0] := 2.96500E+04; afAl[993, 1] := 1.68882E-02;
afAl[994, 0] := 2.97000E+04; afAl[994, 1] := 1.68275E-02;
afAl[995, 0] := 2.97500E+04; afAl[995, 1] := 1.67670E-02;
afAl[996, 0] := 2.98000E+04; afAl[996, 1] := 1.67068E-02;
afAl[997, 0] := 2.98500E+04; afAl[997, 1] := 1.66469E-02;
afAl[998, 0] := 2.99000E+04; afAl[998, 1] := 1.65874E-02;
afAl[999, 0] := 2.99500E+04; afAl[999, 1] := 1.65281E-02;

// Element = Si

